// TIA Portal V21 export
FUNCTION "Motore_AspiratorePompaPistoni" : Void   // FC131, LAD
{ S7_Optimized_Access := 'TRUE' }
// stored: SetENOAutomatically false
   VAR_TEMP
      AutoPos : Bool;
      AutoNeg : Bool;
   END_VAR
BEGIN

REGION Network 1: Comando positivo in automatico
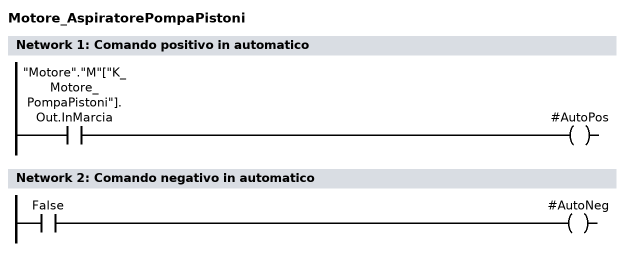
   RUNG wire#powerrail
      Contact( "Motore"."M"["K_Motore_PompaPistoni"].Out.InMarcia )
      Coil( #AutoPos )
   END_RUNG
   // the same network as SCL:
   #AutoPos := "Motore"."M"["K_Motore_PompaPistoni"].Out.InMarcia;
END_REGION

REGION Network 2: Comando negativo in automatico
   RUNG wire#powerrail
      Contact( False )
      Coil( #AutoNeg )
   END_RUNG
   // the same network as SCL:
   #AutoNeg := False;
END_REGION

REGION Network 3 (SCL)
   REGION Aspiratore pompa pistoni
       REGION Ingressi
           "Motore".M[K_Motore_AspiratorePompaPistoni].In.FbDigitali.TermicoIntervenuto := NOT "PompaPistoni_Aspiratore_TermicoOk";
           "Motore".M[K_Motore_AspiratorePompaPistoni].In.FbDigitali.FeedbackMarcia := "PompaPistoni_Aspiratore_Marcia";
           // "Motore".M["K_Motore_AspiratorePompaPistoni"].In.CmdPosRich := #AutoPos;
           // "Motore".M["K_Motore_AspiratorePompaPistoni"].In.CmdNegRich := #AutoNeg;
       END_REGION ;
       REGION Gestione
           "GestMotore"(K_Motore := "K_Motore_AspiratorePompaPistoni",
                        K_TipoMotore := "K_TipoMotore_Teleruttore1Dir",
                        K_Zona := "K_Zona_Sterilizzatore");
       END_REGION ;
       REGION Uscite
           "PompaPistoni_Aspiratore_Marcia" := "Motore".M[K_Motore_AspiratorePompaPistoni].Out.CmdPosMotore;
       END_REGION ;
   END_REGION ;
END_REGION
END_FUNCTION
